FUNCTION_BLOCK Cylinder 
VAR_INPUT
END_VAR
VAR_OUTPUT
	bExtended : BOOL;
	bExtend : BOOL;
END_VAR
VAR
	fbExtendedSignal : BoolIn;
	fbExtend : BoolOut;
END_VAR

bExtended := fbExtendedSignal.getValue;
bExtend := fbExtend.getValue;

METHOD Extend : BOOL
VAR_INPUT
END_VAR
fbExtend.setValue := TRUE;
END_METHOD

PROPERTY getExtend : I_StepCondition
GET
getExtend := fbExtend;
END_GET
END_PROPERTY

METHOD Retract : BOOL
VAR_INPUT
END_VAR
fbExtend.setValue := FALSE;
END_METHOD

END_FUNCTION_BLOCK

(* stored: Version 1.1.0.1, ProductVersion 3.1.4024.2
   POU Cylinder: Id {db89b387-a330-4ef1-99df-108de492603e}, SpecialFunc None
   Method Extend: Id {94bdcdf1-c7f4-49dd-b22c-ac7a00277afb}
   Property getExtend: Id {2b86f911-1673-4bb0-9c31-46cc468eb761}
   Get Get: Id {43470125-c179-4fda-9a24-0ad3f32b4aba}
   Method Retract: Id {4d7b229f-5286-46f1-923f-5cc3f4a39fec} *)
